FUNCTION Greater_Smaller
VAR_INPUT
	nNumber1 : INT;
	nNumber2 : INT;
END_VAR
VAR_OUTPUT
	nGreater : INT;
	nSmaller : INT;
END_VAR

IF nNumber1 > nNumber2 THEN
	nGreater := nNumber1;
	nSmaller := nNumber2;
ELSE
	nGreater := nNumber2;
	nSmaller := nNumber1;	
END_IF

END_FUNCTION

(* stored: Version 1.1.0.1, ProductVersion 3.1.4024.12
   POU Greater_Smaller: Id {c9e68c0e-d2e7-4de5-82c1-7e32ce6d2ae5}, SpecialFunc None *)
